// TIA Portal V19 export
DATA_BLOCK "DB_WT1"   // DB101
{ S7_Optimized_Access := 'FALSE' }
AUTHOR : MS
// stored: AutoNumber false
   VAR RETAIN
      ANZAHL : Int := 10;   // * max. Anzahl der Befehle DB45 beachten!!
      OFFSET : Int := 180;   // * Beginn der Befehlskette
      LENG : Int := 8;   // * Befehlslänge in Byte
      WT_NR_lang : DInt;   // Warenträger-Nr. lang
      Oberflaeche : Real;   // Oberfläche in dm²
      Korb_Nr : USInt;   // Korbnummer (fest)
      POS : USInt;   // aktuelle Position
      Technologie : Int;   // Technologie Code
      priorisiert : Bool;   // WT ist proorisiert
      in_Anlage : Bool;   // will in die Anlage
      in_Entm : Bool;   // will in die Entmetallisierung
      aus_Anlage : Bool;   // kommt aus der Anlage
      aus_Entm : Bool;   // kommt aus der Entmetallisierung
      Speicher : Bool;   // Speicherprogramm
      FW_Pos : Bool;   // WT befindet sich am FW
      QT_Pos : Bool;   // WT befindet sich im QT
      Auto_Pos : USInt;   // Position für Automatikbetrieb
      Trommel : Bool;   // WT ist eine Trommel
      UT_Anforderung : Bool;   // Trockneranforderung erzeugt aus Befehl"FF"
      Stop : Bool;   // Stopbefehl aktiv
      Nassware : Bool;   // Nassware-Trichter am Entladestand anfordern
      TW_Pos : Bool;   // Warenträger ist noch in seiner Taktwechselposition
      noKorrBefx : Bool;   // Befehlsindex nicht korregieren
      noOPT_WT : Bool;   // kann nicht wie berechnet eingefahren werden
      last_Auto : Bool;   // letzter Umsetzvorgang erfolgte in Automatik
      Ziel_Pos_WT : USInt;   // Zielposition des WT für Korrektur beim Einsetzen
      lngsm_senken : Bool;   // langsam Senken
      lngsm_heben : Bool;   // langsam Heben
      lngsm_Fahrt : Bool;   // langsam Fahren
      WT_nok : Bool;   // Behandlungsfehler
      WT_151 : Bool;
      WT_161 : Bool;
      res226 : Bool;
      res227 : Bool;
      Alt_Befx : USInt;   // Befehlsindex in letzter Automatikposition
      Alt_Bereichstakte : USInt;   // Bereichstakte der letzten Automatikposition
      Alt_TW_Pos : USInt;
      Alt_Verweil : DInt;   // Verweilzeit der letzten Automatikposition
      Fertigzeitpunkt : DInt;   // Systemzeit PC, wann WT voraussichtlich fertig
      Meld_Pos : USInt;   // gemerkte Kollisionposition
      WT_Typ : Byte;   // Warenträgertyp (für die Zuordnung bestimmter Ware)
      End_Ziel_Pos : USInt;   // Zielposition an die der WT
      End_Ziel_QT_Pos : USInt;   // Position die ein verwendeter QT anfahren muß
      KorrPend : Real;   // Korrekturfaktor Pendelzeit
      KorrATZ : Real;   // Korrekturfaktor Abtropfzeit
      P_PNTER : Int;   // Parameter-Pointer
      B_PNTER : Int;   // Befehls-pointer
      SaveExpo : DInt;   // gerettete Expozeit bei Zwangsräumung
      Bereichstakte : USInt;   // Takt die der WT noch im aktuellen Behandlungsbereich verbringen muß
      Variante1 : Byte;
      Variante2 : Byte;
      Variante3 : Byte;
      Variante4 : Byte;
      Variante5 : Byte;
      akt_Ziel : Int;   // aktuelles Ziel aus FB9(FC120)
      akt_CMD : Byte;   // aktueller Befehl
      WT_Kennung : Byte;   // farbliche Markierung für PC
      Speed_Up : Int;
      Speed_Dn : Int;
      Speed_Fahrt : Int;
      resI : Int;
      Aufgabezeitpunkt : DInt;   // Systemzeit PC, wann WT aufgegeben wurde
      RestTakte : Int;   // Resttakte durch die Anlage
      "Name" : String[100];
      Befehl : Array[1..20] of Struct   // * Feldlänge anpassen DB45 beachten!!
         Kennung : Byte;   // Befehlskennung
         Startpos : Byte;   // Position
         Laenge : Byte;   // Länge
         Startpos2 : Byte;
         Laenge2 : Byte;
         Sonderparam : Byte;
         Param_Ptr : Int;   // Pointer für Parameter
      END_STRUCT;
      Param_Bereich : Array[1..100] of Byte;   // * Feldlänge anpassen DB45 beachten!!
   END_VAR
BEGIN
END_DATA_BLOCK
